{attribute 'qualified_only'}
{attribute 'strict'}
TYPE Enum_EPT :
(
	eBlocked := 0,
	eIdle,
	eBusy
);
END_TYPE

(* stored: Version 1.1.0.1, ProductVersion 3.1.4022.18
   DUT Enum_EPT: Id {bce93e29-b368-4bc3-8a18-e126a0b1370a} *)
